// TwinCAT 3 PLC project PLC1
// ProgramVersion: 3.1.4022.7
// libraries:
//   Tc2_Standard, * (Beckhoff Automation GmbH)
//   Tc2_System, * (Beckhoff Automation GmbH)
//   Tc3_Module, * (Beckhoff Automation GmbH)
// project tree:
//   / ClassDiagram.TcCD (not stored), PlcTask.TcTTO
//   FBs/Base Class/ FB_Pizza.TcPOU
//   FBs/Sub Classes/ FB_PepperoniPizza.TcPOU, FB_VeggiePizza.TcPOU
//   POUs/ MAIN.TcPOU
// real-time tasks:
//   TASK PlcTask: cycle T#10ms, priority 20, ADS port 350

CONFIGURATION PLC1
    RESOURCE PLC ON TwinCAT3
        TASK PlcTask(INTERVAL := T#10ms, PRIORITY := 20);
        PROGRAM MAIN WITH PlcTask : MAIN;
    END_RESOURCE
END_CONFIGURATION

// ---- POUs/MAIN.TcPOU
PROGRAM MAIN
VAR
	fbPepPizza 	: FB_PepperoniPizza;
	fbVegPizza 	: FB_VeggiePizza;
	
	bPepButton: BOOL;
	bVegButton: BOOL;
END_VAR

fbPepPizza.makePizza(bPepButton);
fbVegPizza.makePizza(bVegButton);

END_PROGRAM

// ---- FBs/Sub Classes/FB_PepperoniPizza.TcPOU
FUNCTION_BLOCK FB_PepperoniPizza EXTENDS FB_Pizza
VAR_INPUT
END_VAR
VAR_OUTPUT
END_VAR
VAR
END_VAR

METHOD addCheese
VAR_INPUT
END_VAR
ADSLOGSTR( msgCtrlMask := ADSLOG_MSGTYPE_WARN,
        	msgFmtStr := 'Adding Mozzarella Cheese...', '');
END_METHOD

METHOD addMeat
VAR_INPUT
END_VAR
ADSLOGSTR( msgCtrlMask := ADSLOG_MSGTYPE_WARN,
        	msgFmtStr := 'Adding Pepperoni...', '');
END_METHOD

METHOD addVegetables : BOOL
VAR_INPUT
END_VAR
// Nothing here because it's not used
// Normally these Meat, Cheese, and Veg would be an Abstract Method
END_METHOD

METHOD customerWantsCheese : BOOL
VAR_INPUT
END_VAR
// Cheese Hook
customerWantsCheese := TRUE;
END_METHOD

METHOD customerWantsMeat : BOOL
VAR_INPUT
END_VAR
// Meat Hook
customerWantsMeat := TRUE;
END_METHOD

END_FUNCTION_BLOCK

// ---- FBs/Base Class/FB_Pizza.TcPOU
FUNCTION_BLOCK PUBLIC FB_Pizza
VAR
	_PizzaState: INT;
	tonPizzaTimer : TON;
END_VAR

METHOD addCheese
VAR_INPUT
END_VAR
// Abstract Method
END_METHOD

METHOD addMeat
VAR_INPUT
END_VAR
//Abstract Method
END_METHOD

METHOD addVegetables : BOOL
VAR_INPUT
END_VAR
//Abstract Method
END_METHOD

METHOD bakePizza
VAR_INPUT
END_VAR
ADSLOGSTR( msgCtrlMask := ADSLOG_MSGTYPE_WARN,
        	msgFmtStr := 'Pizza is in the oven, please wait...', '');
END_METHOD

METHOD boxPizza
VAR_INPUT
END_VAR
ADSLOGSTR( msgCtrlMask := ADSLOG_MSGTYPE_WARN,
        	msgFmtStr := 'Pizza Boxed and Ready!!!', '');
END_METHOD

METHOD customerWantsCheese : BOOL
VAR_INPUT
END_VAR
customerWantsCheese := FALSE;
END_METHOD

METHOD customerWantsMeat : BOOL
VAR_INPUT
END_VAR
customerWantsMeat := FALSE;
END_METHOD

METHOD customerWantsVegetables : BOOL
VAR_INPUT
END_VAR
customerWantsVegetables := FALSE;
END_METHOD

METHOD FINAL makePizza
VAR_INPUT
	bExecute: BOOL;
END_VAR
CASE _PizzaState OF
	0: // Mandatory
		tonPizzaTimer(IN := bExecute, PT := T#2S); 
		IF tonPizzaTimer.Q THEN
			tonPizzaTimer(IN := FALSE, PT := T#2S); 
			rollDough();
			_PizzaState := 10;
		END_IF
		
	10: // Optional
		tonPizzaTimer(IN := TRUE, PT := T#2S); 
		IF tonPizzaTimer.Q THEN
			tonPizzaTimer(IN := FALSE, PT := T#2S); 
			IF(customerWantsCheese()) THEN
				addCheese();
			END_IF
			_PizzaState := 20;
		END_IF
		
	20: // Optional
		tonPizzaTimer(IN := TRUE, PT := T#2S); 
		IF tonPizzaTimer.Q THEN
			tonPizzaTimer(IN := FALSE, PT := T#2S); 
			IF(customerWantsMeat()) THEN
				addMeat();
			END_IF
			_PizzaState := 30;
		END_IF
		
	30: // Optional
		tonPizzaTimer(IN := TRUE, PT := T#2S); 
		IF tonPizzaTimer.Q THEN
			tonPizzaTimer(IN := FALSE, PT := T#2S); 
			IF(customerWantsVegetables()) THEN
				addVegetables();
			END_IF
			_PizzaState := 40;
		END_IF
		
	40: // Mandatory
		tonPizzaTimer(IN := TRUE, PT := T#2S);
 
		IF tonPizzaTimer.Q THEN
			tonPizzaTimer(IN := FALSE, PT := T#2S); 
			bakePizza();
			_PizzaState := 100;
		END_IF
		
	100:// Mandatory
		tonPizzaTimer(IN := TRUE, PT := T#2S); 
		
		IF tonPizzaTimer.Q THEN
			tonPizzaTimer(IN := FALSE, PT := T#2S); 
			boxPizza();
			_PizzaState := 0;
		END_IF
END_CASE
END_METHOD

METHOD rollDough
VAR_INPUT
END_VAR
ADSLOGSTR( msgCtrlMask := ADSLOG_MSGTYPE_WARN,
        	msgFmtStr := 'Rolling the Pizza Dough...', '');
END_METHOD

END_FUNCTION_BLOCK

// ---- FBs/Sub Classes/FB_VeggiePizza.TcPOU
FUNCTION_BLOCK FB_VeggiePizza EXTENDS FB_Pizza
VAR_INPUT
END_VAR
VAR_OUTPUT
END_VAR
VAR
END_VAR

METHOD addCheese
VAR_INPUT
END_VAR
ADSLOGSTR( msgCtrlMask := ADSLOG_MSGTYPE_WARN,
        	msgFmtStr := 'Adding Mozzarella Cheese...', '');
END_METHOD

METHOD addMeat
VAR_INPUT
END_VAR
// Nothing here because it's not used
// Normally these Meat, Cheese, and Veg would be an Abstract Method
END_METHOD

METHOD addVegetables : BOOL
VAR_INPUT
END_VAR
ADSLOGSTR( msgCtrlMask := ADSLOG_MSGTYPE_WARN,
        	msgFmtStr := 'Adding Veggies...', '');
END_METHOD

METHOD customerWantsCheese : BOOL
VAR_INPUT
END_VAR
// Cheese Hook
customerWantsCheese := TRUE;
END_METHOD

METHOD customerWantsVegetables : BOOL
VAR_INPUT
END_VAR
// Veggie Hook
customerWantsVegetables := TRUE;
END_METHOD

END_FUNCTION_BLOCK
